(* IEC 61131-3 sources: Idecon_CheckWeigher_WP/05_Programs, 3 files *)

(* ---- Management_Checkweigher_Idecon.st ---- *)
// ==============================================================================
// Management_Checkweigher_Idecon
// ==============================================================================

// --- 1. RESET INIZIALE E DISABILITAZIONE ---

IF NOT Enable THEN
    Connected := FALSE;
    iRcvState := 0;
    iTestState := 0;
    RxChunkLen := 0;
    RxChunkValid := FALSE;
    TxConsumed := FALSE;
    Command := '';
    CommandTrigger := FALSE;
    G_Idecon_HMI_Cmd.SendTrigger := FALSE;
    G_Test_Ejector_Start := FALSE;
    G_Test_Ejector_Restore := FALSE;
    prevHmiSend := FALSE;
    tonReconnect(IN := FALSE);

    stepInit := 0;
    bInitCloseDone := FALSE;

    fbTcpConnect(Execute := FALSE);
    fbClose(Execute := FALSE);

    RETURN;
END_IF;

// --- 2. SEQUENZA DI INIZIALIZZAZIONE SICURA ---

CASE stepInit OF
    0:
        fbClose(Execute := FALSE, Socket := SocketID_Int);
        stepInit := 10;

    10:
        fbClose(Execute := TRUE, Socket := SocketID_Int);
        IF fbClose.Done OR fbClose.Error THEN
            fbClose(Execute := FALSE, Socket := SocketID_Int);
            stepInit := 20;
        END_IF;

    20:
        bInitCloseDone := TRUE;
END_CASE;

IF NOT bInitCloseDone THEN RETURN; END_IF;

// --- 3. GESTIONE CONNESSIONE TCP ---

tmpIpAddress := Config.IpAdr;
tmpPort := Config.PortNo;

tonReconnect(IN := (NOT Connected AND bConnectError), PT := T#5S);
bEnableConnect := (Enable AND NOT Connected AND NOT bConnectError) OR tonReconnect.Q;

fbTcpConnect(
    Execute     := bEnableConnect,
    DstAdr      := tmpIpAddress,
    DstTcpPort  := tmpPort,
    SrcTcpPort  := 0,
    Socket      => SocketID_Int,
    Done        => bConnectDone,
    Busy        => bConnectBusy,
    Error       => bConnectError,
    ErrorID     => wConnectErrorID
);

IF bConnectDone THEN Connected := TRUE; END_IF;
IF bConnectError THEN Connected := FALSE; END_IF;

// --- 4. MACCHINA A STATI RICEZIONE ---

IF NOT Connected THEN
    iRcvState := 0;
    bExecuteRcv := FALSE;
    iTestState := 0;
END_IF;

CASE iRcvState OF
    0: // IDLE
        IF Connected AND NOT bRcvBusy AND NOT bRcvError THEN
            bExecuteRcv := TRUE;
            iRcvState := 10;
        END_IF;

    10: // WAIT
        IF bRcvDone THEN iRcvState := 20;
        ELSIF bRcvError THEN iRcvState := 20; END_IF;

    20: // RESET
        bExecuteRcv := FALSE;
        IF NOT bRcvDone AND NOT bRcvBusy THEN iRcvState := 0; END_IF;
END_CASE;

fbSocketRcv(
    Execute := bExecuteRcv,
    Socket  := SocketID_Int,
    TimeOut := 1,
    Size    := UINT#512,
    RcvDat  := RxChunk[0],
    Done    => bRcvDone,
    Busy    => bRcvBusy,
    Error   => bRcvError,
    ErrorID => wRcvErrorID,
    RcvSize => RxChunkLen
);

rTrigValid(CLK := (iRcvState = 20) AND (RxChunkLen > 0) AND NOT bRcvError);
RxChunkValid := rTrigValid.Q;

// --- 5. GESTIONE PRIORITÀ COMANDI ---

CommandTrigger := FALSE;

// --- RECUPERO NOME RICETTA ---

sCurrentRecipe := G_Idecon_LastWeight.RecipeName;
IF sCurrentRecipe = '' THEN sCurrentRecipe := G_Idecon_StatP.RecipeName; END_IF;
IF sCurrentRecipe = '' THEN sCurrentRecipe := '400 g'; END_IF; // Fallback

G_Test_Ejector_State := iTestState;

// Timeout di sicurezza per sbloccare lo stato 10 se la bilancia non risponde

tonTestTimeout(IN := (iTestState = 10), PT := T#5S);
IF tonTestTimeout.Q THEN
    iTestState := 0; // Abortisci test per timeout
    G_Test_Ejector_Start := FALSE;
END_IF;

CASE iTestState OF
    0: // IDLE
        IF G_Test_Ejector_Start THEN
            // Passo 1: Leggi config
            Command := CONCAT('GETFROMRECIPE=', CONCAT(sCurrentRecipe, '|EJECTOR_1'));
            CommandTrigger := TRUE;
            pollResetSV := TRUE; pollResetP := TRUE;
            tonPollingSTATSV(IN := FALSE); tonPollingSTATP(IN := FALSE);
            iTestState := 10;
            G_Test_Ejector_Start := FALSE;
        END_IF;

    10: // WAIT READ (Gestito in Parsing e Timeout)

    15: // READ OK -> DISABILITA
        // Passo 2: Disabilita (Offset=0, Durata=0)
        Command := CONCAT('ALTERRECIPE=', CONCAT(sCurrentRecipe, '|EJECTOR_1|0|0'));
        CommandTrigger := TRUE;
        iTestState := 20;

    20: // TESTING
        IF G_Test_Ejector_Restore THEN
            // Passo 3: Ripristina
            Command := CONCAT('ALTERRECIPE=', CONCAT(sCurrentRecipe, '|EJECTOR_1|'));
            Command := CONCAT(Command, G_Test_Saved_Offset);
            Command := CONCAT(Command, '|');
            Command := CONCAT(Command, G_Test_Saved_Duration);
            CommandTrigger := TRUE;
            G_Test_Ejector_Restore := FALSE;
            iTestState := 0;
        END_IF;
END_CASE;

IF (iTestState = 0) OR (iTestState = 20) THEN

    // A. COMANDO MANUALE
    IF G_Idecon_HMI_Cmd.SendTrigger AND NOT prevHmiSend AND NOT CommandTrigger THEN
        Command := G_Idecon_HMI_Cmd.CmdString;
        CommandTrigger := TRUE;
        pollResetSV := TRUE; pollResetP := TRUE;
        tonPollingSTATSV(IN := FALSE); tonPollingSTATP(IN := FALSE);
        G_Idecon_HMI_Cmd.SendTrigger := FALSE;
    END_IF;
    prevHmiSend := G_Idecon_HMI_Cmd.SendTrigger;

    // B. POLLING
    IF NOT CommandTrigger AND (iTestState = 0) AND NOT G_Idecon_HMI_Cmd.SendTrigger THEN
        tonPollingSTATSV(IN := (Enable AND Connected AND NOT pollResetSV), PT := T#2S);
        tonPollingSTATP(IN := (Enable AND Connected AND NOT pollResetP), PT := T#5S);

        pollResetSV := FALSE; pollResetP := FALSE;

        IF tonPollingSTATSV.Q AND NOT prevPollSVQ THEN
            Command := 'STATSV'; CommandTrigger := TRUE; pollResetSV := TRUE;
        ELSIF tonPollingSTATP.Q AND NOT prevPollPQ THEN
            Command := 'STATREQ'; CommandTrigger := TRUE; pollResetP := TRUE;
        END_IF;
        prevPollSVQ := tonPollingSTATSV.Q; prevPollPQ := tonPollingSTATP.Q;
    END_IF;
END_IF;

// --- 6. CHIAMATA DRIVER ---

Idecon(
    Enable := Enable,
    MsgFilter := MsgFilter,
    RxIn := RxChunk,
    RxInLen := RxChunkLen,
    RxInValid := RxChunkValid,
    TxConsumed := TxConsumed,
    Command := Command,
    CommandTrigger := CommandTrigger
);

// --- 7. PARSING RISPOSTE ---

newMsg := (Idecon.LastMessage <> prevLastMessage);
prevLastMessage := Idecon.LastMessage;

IF newMsg THEN
    sTempParse := Idecon.LastMessage;

    // --- PARSING ROBUSTO PER TEST EIETTORE (CORRETTO) ---
    // Se siamo nello stato di attesa risposta (10)
    IF (iTestState = 10) THEN
        // Controlla se è un messaggio di risposta a GETFROMRECIPE
        IF IDECON_StartsWith(sTempParse, 'GETFROMRECIPE=') THEN
            // Rimuovi prefisso: 'GETFROMRECIPE=' (14 char)
            sTempParse := DELETE(sTempParse, 14, 1);

            // --- FIX ROBUSTEZZA: NON controlliamo il campo 2 ---
            // Prendiamo direttamente i valori nei campi 3 e 4.
            // Se sono validi, avanziamo.

            G_Test_Saved_Offset   := IDECON_FieldAt(sTempParse, 3, '|');
            G_Test_Saved_Duration := IDECON_FieldAt(sTempParse, 4, '|');

            // Se abbiamo letto qualcosa di valido, procediamo
            IF (G_Test_Saved_Offset <> '') OR (G_Test_Saved_Duration <> '') THEN
                iTestState := 15; // Successo! Vai allo step successivo
            END_IF;
        END_IF;
    END_IF;

    // --- PARSING STANDARD ---
    newWeightMsg := IDECON_StartsWith(Idecon.LastMessage, 'WEIGHT=');
    IF newWeightMsg AND NOT prevWeightMsg THEN
        G_ProgressiveID := G_ProgressiveID + 1;
    END_IF;
    prevWeightMsg := newWeightMsg;
END_IF;

// --- 8. MAPPATURA OUTPUT ---

tmpWeightData := Idecon.Weight;
tmpStatPData  := Idecon.StatP;
G_Idecon_LastSTATSV := Idecon.LastSTATSV;

IF tmpWeightData.Valid THEN G_Idecon_LastWeight := tmpWeightData; G_Idecon_LastWeight.Valid := TRUE; END_IF;
IF tmpStatPData.Valid THEN G_Idecon_StatP := tmpStatPData; G_Idecon_StatP.Valid := TRUE; END_IF;

// --- 9. ERRORI E OPC UA ---

G_System_Error := bConnectError OR bSendError OR bRcvError OR Idecon.Error;

IF G_Idecon_StatP.Valid AND (G_Idecon_StatP.TotalProducts >= G_Idecon_StatP.TotalAccepted) THEN
    totalRejected := G_Idecon_StatP.TotalProducts - G_Idecon_StatP.TotalAccepted;
ELSE totalRejected := 0; END_IF;

// Mapping OPC UA

G_OPCUA_Idecon.Connected := Connected;
G_OPCUA_Idecon.WorkMode := G_Idecon_WorkMode;
G_OPCUA_Idecon.LastSTATSV := G_Idecon_LastSTATSV;
G_OPCUA_Idecon.BatchCode := G_Idecon_BatchCode;
G_OPCUA_Idecon.ProductionOrder := G_Idecon_ProductionOrder;
G_OPCUA_Idecon.Error := G_System_Error;
G_OPCUA_Idecon.ErrorId := UINT_TO_UDINT(WORD_TO_UINT(wConnectErrorID));

G_OPCUA_Idecon.LastWeight.ProgressiveId := G_ProgressiveID;
G_OPCUA_Idecon.LastWeight.TimestampText := G_Idecon_LastWeight.DateTimeText;
G_OPCUA_Idecon.LastWeight.ProductionOrder := G_Idecon_LastWeight.ProductionOrder;
G_OPCUA_Idecon.LastWeight.BatchCode := G_Idecon_LastWeight.BatchCode;
G_OPCUA_Idecon.LastWeight.RecipeName := G_Idecon_LastWeight.RecipeName;
G_OPCUA_Idecon.LastWeight.LineCode := G_Idecon_LastWeight.LineCode;
G_OPCUA_Idecon.LastWeight.SerialNumber := G_Idecon_LastWeight.SerialNumber;
G_OPCUA_Idecon.LastWeight.Weight_g := DINT_TO_LREAL(G_Idecon_LastWeight.WeightMg) / LREAL#1000.0;
G_OPCUA_Idecon.LastWeight.Delta_g := DINT_TO_LREAL(G_Idecon_LastWeight.DeltaToNominalMg) / LREAL#1000.0;
G_OPCUA_Idecon.LastWeight.Classification := G_Idecon_LastWeight.Classification;
// FIX ESPULSIONE: Controllo Bit 8 (Expelled Generico) o Bit 15 (Expelled per Consenso)
// Usiamo la conversione esplicita per evitare errori di sintassi
G_OPCUA_Idecon.LastWeight.Expelled := ((G_Idecon_LastWeight.Classification AND DWORD#16#100) > DWORD#0) OR
                                      ((G_Idecon_LastWeight.Classification AND DWORD#16#8000) > DWORD#0);
G_OPCUA_Idecon.LastWeight.Valid := G_Idecon_LastWeight.Valid;

G_OPCUA_Idecon.Stats.TotalProducts := G_Idecon_StatP.TotalProducts;
G_OPCUA_Idecon.Stats.TotalAccepted := G_Idecon_StatP.TotalAccepted;
G_OPCUA_Idecon.Stats.TotalRejected := totalRejected;
G_OPCUA_Idecon.Stats.RejectedPlusPlus := G_Idecon_StatP.RejectedPlusPlus;
G_OPCUA_Idecon.Stats.CannotBeWeighed := G_Idecon_StatP.CannotBeWeighed;
G_OPCUA_Idecon.Stats.MetalCategory := G_Idecon_StatP.MetalCategory;
G_OPCUA_Idecon.Stats.Valid := G_Idecon_StatP.Valid;

// --- 10. INVIO SOCKET ---

sendTrigger := (Idecon.TxOutValid AND NOT prevTxOutValid);
prevTxOutValid := Idecon.TxOutValid;

IF sendTrigger THEN TxBuffer := Idecon.TxOut; END_IF;

fbSocketSend(
    Execute := (Enable AND Connected AND sendTrigger),
    Socket := SocketID_Int,
    SendDat := TxBuffer[0],
    Size := Idecon.TxOutLen,
    Done => bSendDone,
    Busy => bSendBusy,
    Error => bSendError,
    ErrorID => wSendErrorID
);
TxConsumed := bSendDone;

IF NOT Enable AND Connected THEN
    fbClose(Execute := TRUE, Socket := SocketID_Int);
ELSE
    fbClose(Execute := FALSE, Socket := SocketID_Int);
END_IF;

(* ---- Test_Idecon_Connection.st ---- *)
// ==============================================================================
// TEST: Idecon_ConnectionTest
// DESCRIZIONE: Test di connessione alla pesatrice IDECON
// IP: 172.16.224.210 | Port: 50000
// ==============================================================================

VAR
    // TCP Connection
    fbTcpConnect : SysSocketConnect;
    fbSocketRcv : SysSocketRcv;
    fbSocketSend : SysSocketSend;
    fbClose : SysSocketClose;

    // Status
    SocketID : UDINT;
    Connected : BOOL;
    bConnectBusy : BOOL;
    bConnectDone : BOOL;
    bConnectError : BOOL;
    wConnectErrorID : WORD;
    bRcvDone : BOOL;
    bRcvBusy : BOOL;
    bRcvError : BOOL;
    wRcvErrorID : WORD;
    bSendDone : BOOL;
    bSendBusy : BOOL;
    bSendError : BOOL;
    wSendErrorID : WORD;

    // RX/TX Buffers
    RxBuf : ARRAY[0..511] OF BYTE;
    RxLen : UINT;
    TxBuf : ARRAY[0..255] OF BYTE;
    TxLen : UINT;

    // Test Control
    TestEnable : BOOL;
    TestStep : INT;
    tonReceive : TON;
    tonConnect : TON;
    ResultMessage : STRING[255];
    ConnectionStatus : STRING[50];

    // Received Data
    ReceivedString : STRING[512];
    ResponseCount : UDINT;
END_VAR

// ==============================================================================
// MAIN TEST LOGIC
// ==============================================================================

IF NOT TestEnable THEN
    // Reset
    Connected := FALSE;
    TestStep := 0;
    ResponseCount := 0;
    ReceivedString := '';
    ConnectionStatus := 'Idle';
    ResultMessage := '';

    fbTcpConnect(Execute := FALSE);
    fbSocketRcv(Execute := FALSE);
    fbSocketSend(Execute := FALSE);
    fbClose(Execute := FALSE);

    RETURN;
END_IF;

// Connection Timeout (10 seconds)
tonConnect(IN := TestEnable, PT := T#10S);
IF tonConnect.Q THEN
    ConnectionStatus := 'Timeout - No Connection';
    TestStep := 100; // Error state
END_IF;

// Receive Timeout (3 seconds per command)
tonReceive(IN := (TestStep = 20), PT := T#3S);
IF tonReceive.Q THEN
    ConnectionStatus := 'Timeout - No Response';
    TestStep := 100;
END_IF;

// State Machine
CASE TestStep OF
    0: // Connect
        ConnectionStatus := 'Connecting...';
        fbTcpConnect(
            Execute := TRUE,
            DstAdr := '172.16.224.210',
            DstTcpPort := 50000,
            SrcTcpPort := 0,
            Socket => SocketID,
            Done => bConnectDone,
            Busy => bConnectBusy,
            Error => bConnectError,
            ErrorID => wConnectErrorID
        );

        IF bConnectDone THEN
            Connected := TRUE;
            TestStep := 10;
            ConnectionStatus := 'Connected!';
        ELSIF bConnectError THEN
            ConnectionStatus := CONCAT('Connect Error: ', UINT_TO_STRING(wConnectErrorID));
            TestStep := 100;
        END_IF;

    10: // Start Receiving
        fbTcpConnect(Execute := FALSE);
        ConnectionStatus := 'Waiting for data...';
        TestStep := 20;

    20: // Receive Loop
        fbSocketRcv(
            Execute := TRUE,
            Socket := SocketID,
            TimeOut := 1,
            Size := 512,
            RcvDat => RxBuf[0],
            Done => bRcvDone,
            Busy => bRcvBusy,
            Error => bRcvError,
            ErrorID => wRcvErrorID,
            RcvSize => RxLen
        );

        IF bRcvDone AND RxLen > 0 THEN
            // Process received data
            fbSocketRcv(Execute := FALSE);

            // Convert bytes to string for display
            ReceivedString := '';
            FOR i := 0 TO INT_TO_UINT(RxLen - 1) DO
                IF RxBuf[i] >= 32 AND RxBuf[i] <= 126 THEN
                    ReceivedString := CONCAT(ReceivedString, BYTE_TO_CHAR(RxBuf[i]));
                ELSE
                    ReceivedString := CONCAT(ReceivedString, '.');
                END_IF;
            END_FOR;

            ResponseCount := ResponseCount + 1;
            ConnectionStatus := CONCAT('Data Received (', UINT_TO_STRING(ResponseCount), ')');

            // Send STATSV command to test
            TestStep := 30;
        ELSIF bRcvError THEN
            ConnectionStatus := 'Receive Error';
            TestStep := 100;
        END_IF;

    30: // Send STATSV Command
        // Prepare STATSV command: STX + 'STATSV' + ETX
        TxBuf[0] := 16#02;  // STX
        TxBuf[1] := 16#53;  // S
        TxBuf[2] := 16#54;  // T
        TxBuf[3] := 16#41;  // A
        TxBuf[4] := 16#54;  // T
        TxBuf[5] := 16#53;  // S
        TxBuf[6] := 16#56;  // V
        TxBuf[7] := 16#03;  // ETX
        TxLen := 8;

        fbSocketSend(
            Execute := TRUE,
            Socket := SocketID,
            SendDat => TxBuf[0],
            Size := TxLen,
            Done => bSendDone,
            Busy => bSendBusy,
            Error => bSendError,
            ErrorID => wSendErrorID
        );

        IF bSendDone THEN
            ResultMessage := 'STATSV Command Sent';
            TestStep := 20; // Back to receive
        ELSIF bSendError THEN
            ConnectionStatus := 'Send Error';
            TestStep := 100;
        END_IF;

    100: // Error / Cleanup
        ResultMessage := 'Test Ended with Error';

    200: // Disconnect
        fbClose(Execute := TRUE, Socket := SocketID);
        IF fbClose.Done THEN
            Connected := FALSE;
            TestEnable := FALSE;
            ConnectionStatus := 'Disconnected';
        END_IF;
END_CASE;

// Auto-stop after 30 seconds of successful connection
IF TestStep = 20 AND TestEnable THEN
    // Keep receiving...
END_IF;

(* ---- Var_Management_Checkweigher_Idecon.st ---- *)
VAR Internal
tmpIpAddress	STRING[256]			False	False
Config	_sSOCKET_ADDRESS	(PortNo := 50000, IpAdr := '172.16.224.200')		False	False
tmpPort	UINT			False	False
bConnectError	BOOL			False	False
bEnableConnect	BOOL			False	False
bConnectDone	BOOL			False	False
bConnectBusy	BOOL			False	False
wConnectErrorID	WORD			False	False
bExecuteRcv	BOOL			False	False
bRcvBusy	BOOL			False	False
bRcvError	BOOL			False	False
bRcvDone	BOOL			False	False
fbSocketRcv	SktTCPRcv			False	False
RxChunk	ARRAY[0..511] OF BYTE			False	False
wRcvErrorID	WORD			False	False
rTrigValid	R_TRIG			False	False
sCurrentRecipe	STRING[64]			False	False
tonTestTimeout	TON			False	False
pollResetSV	BOOL			False	False
pollResetP	BOOL			False	False
tonPollingSTATSV	TON			False	False
tonPollingSTATP	TON			False	False
prevPollSVQ	BOOL			False	False
prevPollPQ	BOOL			False	False
Idecon	FB_IDECON_Client			False	False
MsgFilter	UINT	17		False	False
newMsg	BOOL			False	False
prevLastMessage	STRING[512]			False	False
sTempParse	STRING[255]			False	False
newWeightMsg	BOOL			False	False
prevWeightMsg	BOOL			False	False
tmpWeightData	Idecon_WeightData			False	False
tmpStatPData	Idecon_StatPData			False	False
bSendError	BOOL			False	False
totalRejected	DINT			False	False
sendTrigger	BOOL			False	False
prevTxOutValid	BOOL			False	False
TxBuffer	ARRAY[0..511] OF BYTE			False	False
fbSocketSend	SktTCPSend			False	False
bSendDone	BOOL			False	False
bSendBusy	BOOL			False	False
wSendErrorID	WORD			False	False
END_VAR

VAR External
HMI_MachineSetUp	False
HMI_OnLineData	False
FLAG	False
HMI_OnlineStatistics	False
SEQUENCE	False
HMI_NoRecipeMachine	False
AXIS	False
ScadaInterface	False
MachineAnalytics	False
HMI_RecipeMachine	False
HMI_RecipeName	False
D_Recipes	False
RecipeArchives	False
TimeZoneAndDLS_DateTime	False
ScadaLogs	False
G_Idecon_HMI_Cmd	False
G_Test_Ejector_Start	False
G_Test_Ejector_Restore	False
G_Idecon_LastWeight	False
G_Idecon_StatP	False
G_Test_Ejector_State	False
G_Test_Saved_Offset	False
G_Test_Saved_Duration	False
G_ProgressiveID	False
G_Idecon_LastSTATSV	False
G_System_Error	False
G_OPCUA_Idecon	False
G_Idecon_WorkMode	False
G_Idecon_BatchCode	False
G_Idecon_ProductionOrder	False

.
